(* IEC 61131-3 sources: ICSQuartz/benchmarks/oscat_basic_del_chars/src, 1 file *)

(* ---- program.st ---- *)
PROGRAM PLC_PRG
VAR_INPUT
    in_in: STRING;
    in_cx: STRING;
END_VAR

DEL_CHARS(in_in, in_cx);

END_PROGRAM
